{attribute 'GeneratedUsingTerminal: EK1122-0000-0018'}
{attribute addProperty BoxType "EK1122-0000-0018"}
{attribute addProperty Id "Beckhoff_EJ5xxxsub_EK1100EK1100_1FC0878B2"}
{attribute addProperty CRC "2821468474"}
{attribute addProperty Size "2"}
TYPE Beckhoff_EJ5xxxEK1122_A82C313A EXTENDS EK1122_1FC0878B :
STRUCT
	{attribute addProperty Name "Beckhoff EJ5xxxsub EK1100"}
	{attribute addProperty PreviousPort "Beckhoff EJ5xxxEK1122 : D"}
	Beckhoff_EJ5xxxsub_EK1100 : EK1100_1FC0878B;
END_STRUCT
END_TYPE

(* stored: Version 1.2.0.0, ProductVersion 3.1.4024.11
   DUT Beckhoff_EJ5xxxEK1122_A82C313A: Id {1a39befd-857b-4c9f-ba37-a93114a59673} *)
